PROGRAM Disconnect
VAR
	Disconnect_R1			:FB_Trennen;
	Disconnect_R2			:FB_Trennen;
	Disconnect_R3			:FB_Trennen;
	Disconnect_R4			:FB_Trennen;
	Disconnect_R5			:FB_Trennen;
	Disconnect_R6			:FB_Trennen;
	Disconnect_R7			:FB_Trennen;
END_VAR

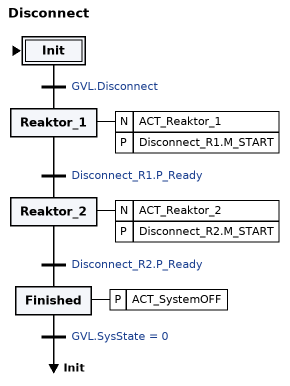
INITIAL_STEP Init:
END_STEP
TRANSITION FROM Init TO Reaktor_1
    := GVL.Disconnect;
END_TRANSITION
STEP Reaktor_1:
    ACT_Reaktor_1(N);
    Disconnect_R1.M_START(P);
END_STEP
TRANSITION FROM Reaktor_1 TO Reaktor_2
    := Disconnect_R1.P_Ready;
END_TRANSITION
STEP Reaktor_2:
    ACT_Reaktor_2(N);
    Disconnect_R2.M_START(P);
END_STEP
TRANSITION FROM Reaktor_2 TO Finished
    := Disconnect_R2.P_Ready;
END_TRANSITION
STEP Finished:
    ACT_SystemOFF(P);
END_STEP
TRANSITION FROM Finished TO Init
    := GVL.SysState = 0;
END_TRANSITION

ACTION ACT_Reaktor_1:
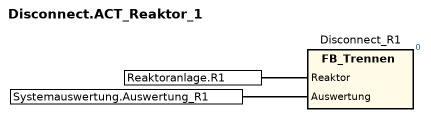
Disconnect_R1(Reaktor := Reaktoranlage.R1, Auswertung := Systemauswertung.Auswertung_R1); // FB_Trennen
END_ACTION

ACTION ACT_Reaktor_2:
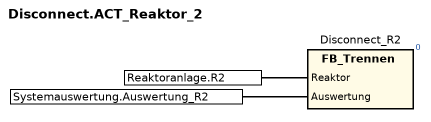
Disconnect_R2(Reaktor := Reaktoranlage.R2, Auswertung := Systemauswertung.Auswertung_R2); // FB_Trennen
END_ACTION

ACTION ACT_SystemOFF:
GVL.SysState := 0;
END_ACTION

END_PROGRAM

(* stored: Version 1.1.0.1, ProductVersion 3.1.4024.12
   POU Disconnect: Id {b1c2c0dc-26a4-4ce3-8cf8-1d472f0b3671}, SpecialFunc None
   Action ACT_Reaktor_1: Id {db6d4f86-81a3-453a-8eb0-931c39a196ee}
   Action ACT_Reaktor_2: Id {c2157551-f262-4685-9543-0fea69a2e46c}
   Action ACT_SystemOFF: Id {f9735299-b0cc-40b1-ba62-496a310beb9a} *)
